TYPE EL6022 :
STRUCT
	Channel_1 : EL6022_CHANNEL;
	Channel_2 : EL6022_CHANNEL;
END_STRUCT
END_TYPE

(* stored: Version 1.1.0.1, ProductVersion 3.1.4026.18
   DUT EL6022: Id {3bfb6762-705e-45d9-b3d0-da51074e3bf1} *)
